Yaskawa INFORM job: R2_W73(0'-90)AWOK.JBI

/JOB
//NAME R2_W73(0'-90)AWOK
///FOLDERNAME AWOK
//POS
///NPOS 44,44,0,2,0,0
///TOOL 0
///POSTYPE PULSE
///PULSE
C00000=145854,64802,-7540,-5361,88024,-33305
C00001=146518,67008,-1742,-5685,85636,-33021
C00002=146775,67981,670,-5813,84671,-32906
C00003=149069,69848,3561,-6917,84005,-32228
C00004=148977,68743,3775,-6879,83306,-32216
C00005=149069,69848,3561,-6917,84005,-32228
C00006=146775,67981,670,-5813,84671,-32906
C00007=141709,70505,3632,5716,88123,-35177
C00008=142143,70760,4061,5528,87966,-35063
C00009=141709,70505,3632,5716,88123,-35177
C00010=141466,75678,7759,5822,88256,-35240
C00011=150714,57521,-9985,-12467,84539,-31420
C00012=152043,57091,-7724,-13148,83136,-30899
C00013=151905,57965,-6718,-13084,82951,-30919
C00014=152043,57091,-7724,-13148,83136,-30899
C00015=150714,57521,-9985,-12467,84539,-31420
C00016=149545,64988,-1239,-11917,82883,-31588
C00017=150397,65709,-1678,-12325,83616,-31417
C00018=153374,75160,10795,-20701,82940,-35643
C00019=153562,73111,9572,-20799,82698,-35542
C00020=145671,67847,3957,2275,78950,-48491
C00021=139796,73037,10697,20742,81976,-59006
C00022=139855,76006,10433,20657,83547,-58718
C00023=138944,70547,-13352,-2713,109632,-82660
C00024=150992,69723,-1355,-37332,105967,-89594
C00025=150476,128390,79342,-39456,121713,-63684
C00026=150050,126781,76809,-37795,123285,-66166
C00027=152913,78185,12310,-42752,113213,-84591
C00028=152182,82606,18149,-42190,111927,-84311
C00029=152182,83304,17941,-42342,112294,-84475
C00030=151694,72284,4221,-38531,106791,-89962
C00031=151725,70435,2944,-38503,106671,-89906
C00032=151269,73478,6661,-38228,105932,-89795
C00033=151161,78896,6636,-38820,108108,-90659
C00034=150730,108324,43859,-37200,101741,-88479
C00035=138109,93543,17707,-11473,100978,-85696
C00036=126155,75677,-665,13089,94512,-81960
C00037=136360,44466,-35259,-6214,94815,-84020
C00038=129275,89679,9974,19452,120712,-90755
C00039=124823,94818,27238,29160,120181,-86319
C00040=125815,95145,27666,29078,119805,-86047
C00041=125255,100992,28971,31279,121490,-85312
C00042=115228,95345,30870,-14961,82572,-85130
C00043=91123,51604,-32991,-14961,82572,-85130
BC00000=299173,218396,1075175
BC00001=299173,218396,1075175
BC00002=299173,218396,1075175
BC00003=299173,218396,1075175
BC00004=299173,218396,1075175
BC00005=299173,218396,1075175
BC00006=299173,218396,1075175
BC00007=299173,218396,1075175
BC00008=299173,218396,1075175
BC00009=299173,218396,1075175
BC00010=299173,218396,1075175
BC00011=299173,218396,1075175
BC00012=299173,218396,1075175
BC00013=299173,218396,1075175
BC00014=299173,218396,1075175
BC00015=299173,218396,1075175
BC00016=299173,218396,1075175
BC00017=299173,218396,1075175
BC00018=299173,218396,1075175
BC00019=299173,218396,1075175
BC00020=299173,218396,1075175
BC00021=299173,218396,1075175
BC00022=299173,218396,1075175
BC00023=236130,188559,1075175
BC00024=236130,188559,1075175
BC00025=236130,181604,1075175
BC00026=236130,181604,1075175
BC00027=236130,181604,1075175
BC00028=236130,181604,1075175
BC00029=236130,181604,1075175
BC00030=236130,181604,1075175
BC00031=236130,181604,1075175
BC00032=236130,181604,1075175
BC00033=236130,181604,1075175
BC00034=236130,181604,1075175
BC00035=236130,181604,1075175
BC00036=236130,181604,1075175
BC00037=236130,181604,1075175
BC00038=236130,181604,1075175
BC00039=236130,181604,1075175
BC00040=236130,181604,1075175
BC00041=236130,181604,1075175
BC00042=209008,432171,1075171
BC00043=209008,432171,1075171
///POSTYPE BASE
///RECTAN
///RCONF 0,0,0,0,0,0,0,0,0,0,0,0,0,0,0,0,0,0,0,0,0,0,0,0
P00006=0.222,-3.123,-1.508,0.0000,0.0000,0.0000
P00022=0.222,-3.123,-1.508,0.0000,0.0000,0.0000
//INST
///DATE 2023/11/16 10:50
///ATTR SC,RW
///GROUP1 RB1,BS1
NOP
'r2_W73(search-tylko)
'spawanie na krzyÅ¼
'spawanie na krzyÅ¼
'spawanie na krzyÅ¼
'Path S1141
SFTOF
MOVJ C00000 BC00000 VJ=20.00
MOVL C00001 BC00001 V=100.0
MOVL C00002 BC00002 V=100.0
MOVL C00003 BC00003 V=60.0
REFP 3 C00004 BC00004
CALL JOB:SEARCH-R1
SET P022 P006
SFTON P022
MOVL C00005 BC00005 V=60.0
MOVL C00006 BC00006 V=100.0
MOVL C00007 BC00007 V=60.0
REFP 3 C00008 BC00008
CALL JOB:SEARCH-R1
SET P022 P006
SFTON P022
MOVL C00009 BC00009 V=60.0
MOVL C00010 BC00010 V=100.0
MOVL C00011 BC00011 V=100.0
MOVL C00012 BC00012 V=60.0
REFP 3 C00013 BC00013
CALL JOB:SEARCH-R1
SET P022 P006
SFTON P022
MOVL C00014 BC00014 V=60.0
MOVL C00015 BC00015 V=100.0
MOVL C00016 BC00016 V=100.0
MOVL C00017 BC00017 V=100.0
SFTOF
SFTOF
SFTON P022
MOVL C00018 BC00018 V=100.0
MOVL C00019 BC00019 V=100.0 PL=0
MACRO1 MJ#(0) ARGF9
ARCON
MOVL C00020 BC00020 V=10.8
MOVL C00021 BC00021 V=10.8
ARCOF
MOVL C00022 BC00022 V=100.0
MOVL C00023 BC00023 V=100.0
MOVJ C00024 BC00024 VJ=20.00
'COMMENT
'COMMENT
SFTOF
SFTON P022
MOVL C00025 BC00025 V=100.0
MOVL C00026 BC00026 V=100.0 PL=0
MACRO1 MJ#(0) ARGF9
ARCON
MOVL C00027 BC00027 V=10.8
MOVL C00028 BC00028 V=10.8
ARCOF
MOVL C00029 BC00029 V=100.0
MOVL C00030 BC00030 V=100.0
'COMMENT
'COMMENT
SFTOF
SFTON P022
MOVL C00031 BC00031 V=100.0 PL=0
MACRO1 MJ#(0) ARGF9
ARCON
MOVL C00032 BC00032 V=10.8
ARCOF
MOVL C00033 BC00033 V=100.0
MOVJ C00034 BC00034 VJ=20.00
MOVJ C00035 BC00035 VJ=20.00
MOVJ C00036 BC00036 VJ=20.00
MOVJ C00037 BC00037 VJ=20.00
MOVJ C00038 BC00038 VJ=20.00
'COMMENT
'COMMENT
SFTOF
SFTON P022
MOVL C00039 BC00039 V=100.0 PL=0
MACRO1 MJ#(0) ARGF9
ARCON
MOVL C00040 BC00040 V=10.8
ARCOF
MOVL C00041 BC00041 V=100.0
SFTOF
MOVJ C00042 BC00042 VJ=20.00
MOVJ C00043 BC00043 VJ=20.00
END
